FUNCTION_BLOCK DigitalInput_NC_TEST
VAR
END_VAR

ForcedOn();
ForcedOff();
On();
Off();

METHOD ForcedOff : BOOL
VAR
	Expected		: BOOL;
	Actual			: BOOL;
	Input			: BOOL;
	DigitalInput_NC : DigitalInput_NC('DigitalInput', Input);
END_VAR
IF TestSuite.Test(__POUNAME()).ExecuteTest() THEN
	Expected			  := FALSE;
	DigitalInput_NC.Force := E_ForceState.ForceOff;
	Input				  := FALSE;
	Actual				  := DigitalInput_NC.IsActive;
	TestSuite.Test(__POUNAME()).AssertEqual(Expected, Actual);
END_IF
END_METHOD

METHOD ForcedOn : BOOL
VAR
	Expected		: BOOL;
	Actual			: BOOL;
	Input			: BOOL;
	DigitalInput_NC : DigitalInput_NC('DigitalInput', Input);
END_VAR
IF TestSuite.Test(__POUNAME()).ExecuteTest() THEN
	Expected			  := TRUE;
	DigitalInput_NC.Force := E_ForceState.ForceOn;
	Input				  := TRUE;
	Actual				  := DigitalInput_NC.IsActive;
	TestSuite.Test(__POUNAME()).AssertEqual(Expected, Actual);
END_IF
END_METHOD

METHOD Off : BOOL
VAR
	Expected		: BOOL;
	Actual			: BOOL;
	Input			: BOOL;
	DigitalInput_NC : DigitalInput_NC('DigitalInput', Input);
END_VAR
IF TestSuite.Test(__POUNAME()).ExecuteTest() THEN
	Expected			  := FALSE;
	DigitalInput_NC.Force := E_ForceState.Unforced;
	Input				  := TRUE;
	Actual				  := DigitalInput_NC.IsActive;
	TestSuite.Test(__POUNAME()).AssertEqual(Expected, Actual);
END_IF
END_METHOD

METHOD On
VAR
	Expected		: BOOL;
	Actual			: BOOL;
	Input			: BOOL;
	DigitalInput_NC : DigitalInput_NC('DigitalInput', Input);
END_VAR
IF TestSuite.Test(__POUNAME()).ExecuteTest() THEN
	Expected			  := TRUE;
	DigitalInput_NC.Force := E_ForceState.Unforced;
	Input				  := FALSE;
	Actual				  := DigitalInput_NC.IsActive;
	TestSuite.Test(__POUNAME()).AssertEqual(Expected, Actual);
END_IF
END_METHOD

END_FUNCTION_BLOCK

(* stored: Version 1.1.0.1, ProductVersion 3.1.4026.18
   POU DigitalInput_NC_TEST: Id {e9214884-715e-486d-b6b0-594869346b3c}, SpecialFunc None
   Method ForcedOff: Id {5db2355d-80e2-43b5-8ede-1fa6b7ffb802}
   Method ForcedOn: Id {3cd99017-f14a-42eb-8d24-8a743d6673a9}
   Method Off: Id {899584b3-5dcc-4106-86b6-f9aafeb05755}
   Method On: Id {50df22eb-6301-41fc-9b18-f07dd55bf9a6} *)
